FUNCTION_BLOCK FB_BreakTheArbiter
VAR_INPUT
	
END_VAR
VAR_OUTPUT
END_VAR
VAR
END_VAR

END_FUNCTION_BLOCK

(* stored: Version 1.1.0.1, ProductVersion 3.1.4022.12
   POU FB_BreakTheArbiter: Id {572de4b8-f6c3-0c43-352b-59452dfd0cf0}, SpecialFunc None *)
